// TIA Portal V21 export
FUNCTION "SUBOUT" : Void   // FC16, LAD
{ S7_Optimized_Access := 'TRUE' }
// stored: SetENOAutomatically false
   VAR_TEMP   // added for the SCL form of the ladder/FBD networks
      _w1 : Bool;
      _w2 : Bool;
   END_VAR
BEGIN

REGION Network 1
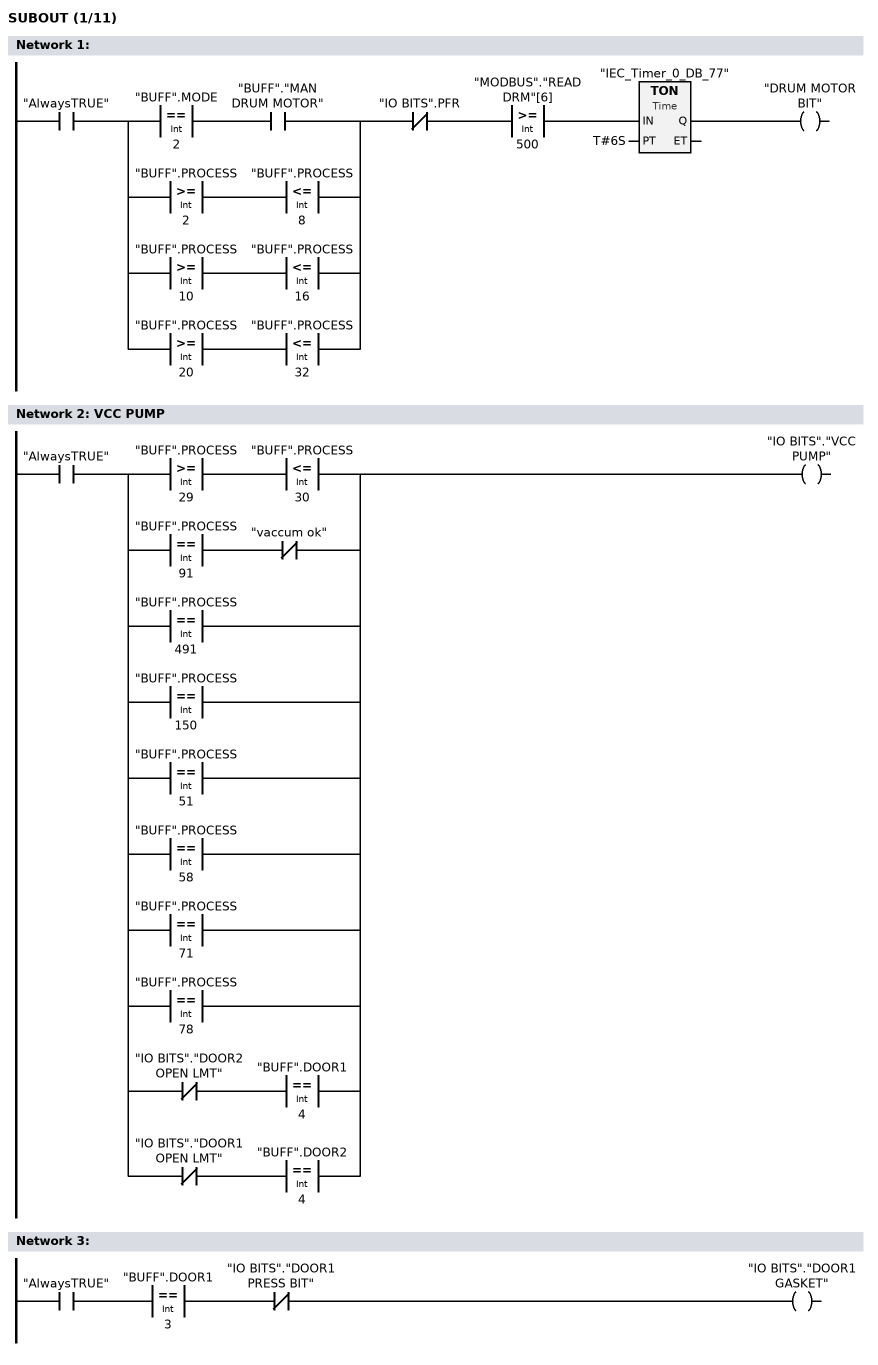
   RUNG wire#powerrail
      Contact( "AlwaysTRUE" )
      wire#w1
      { S7_Templates := "SrcType := Int" } EQ_Contact(in1 := "BUFF".MODE, in2 := 2)
      Contact( "BUFF"."MAN DRUM MOTOR" )
      wire#w2
      I_Contact( "IO BITS".PFR )
      { S7_Templates := "SrcType := Int" } GE_Contact(in1 := "MODBUS"."READ DRM"[6], in2 := 500)
      { S7_Templates := "time_type := Time" } "IEC_Timer_0_DB_77".TON(pt := T#6S, et =>)
      Coil( "DRUM MOTOR BIT" )
   END_RUNG
   RUNG wire#w1
      { S7_Templates := "SrcType := Int" } GE_Contact(in1 := "BUFF".PROCESS, in2 := 2)
      { S7_Templates := "SrcType := Int" } LE_Contact(in1 := "BUFF".PROCESS, in2 := 8)
   END_RUNG wire#w2
   RUNG wire#w1
      { S7_Templates := "SrcType := Int" } GE_Contact(in1 := "BUFF".PROCESS, in2 := 10)
      { S7_Templates := "SrcType := Int" } LE_Contact(in1 := "BUFF".PROCESS, in2 := 16)
   END_RUNG wire#w2
   RUNG wire#w1
      { S7_Templates := "SrcType := Int" } GE_Contact(in1 := "BUFF".PROCESS, in2 := 20)
      { S7_Templates := "SrcType := Int" } LE_Contact(in1 := "BUFF".PROCESS, in2 := 32)
   END_RUNG wire#w2
   // the same network as SCL:
   "IEC_Timer_0_DB_77".TON(IN := "AlwaysTRUE" AND ((("BUFF".MODE = 2) AND "BUFF"."MAN DRUM MOTOR") OR (("BUFF".PROCESS >= 2) AND ("BUFF".PROCESS <= 8)) OR (("BUFF".PROCESS >= 10) AND ("BUFF".PROCESS <= 16)) OR (("BUFF".PROCESS >= 20) AND ("BUFF".PROCESS <= 32))) AND NOT "IO BITS".PFR AND ("MODBUS"."READ DRM"[6] >= 500),
                           PT := T#6S);
   "DRUM MOTOR BIT" := "IEC_Timer_0_DB_77".Q;
END_REGION

REGION Network 2: VCC PUMP
   RUNG wire#powerrail
      Contact( "AlwaysTRUE" )
      wire#w1
      { S7_Templates := "SrcType := Int" } GE_Contact(in1 := "BUFF".PROCESS, in2 := 29)
      { S7_Templates := "SrcType := Int" } LE_Contact(in1 := "BUFF".PROCESS, in2 := 30)
      wire#w2
      Coil( "IO BITS"."VCC PUMP" )
   END_RUNG
   RUNG wire#w1
      { S7_Templates := "SrcType := Int" } EQ_Contact(in1 := "BUFF".PROCESS, in2 := 91)
      I_Contact( "vaccum ok" )
   END_RUNG wire#w2
   RUNG wire#w1
      { S7_Templates := "SrcType := Int" } EQ_Contact(in1 := "BUFF".PROCESS, in2 := 491)
   END_RUNG wire#w2
   RUNG wire#w1
      { S7_Templates := "SrcType := Int" } EQ_Contact(in1 := "BUFF".PROCESS, in2 := 150)
   END_RUNG wire#w2
   RUNG wire#w1
      { S7_Templates := "SrcType := Int" } EQ_Contact(in1 := "BUFF".PROCESS, in2 := 51)
   END_RUNG wire#w2
   RUNG wire#w1
      { S7_Templates := "SrcType := Int" } EQ_Contact(in1 := "BUFF".PROCESS, in2 := 58)
   END_RUNG wire#w2
   RUNG wire#w1
      { S7_Templates := "SrcType := Int" } EQ_Contact(in1 := "BUFF".PROCESS, in2 := 71)
   END_RUNG wire#w2
   RUNG wire#w1
      { S7_Templates := "SrcType := Int" } EQ_Contact(in1 := "BUFF".PROCESS, in2 := 78)
   END_RUNG wire#w2
   RUNG wire#w1
      I_Contact( "IO BITS"."DOOR2 OPEN LMT" )
      { S7_Templates := "SrcType := Int" } EQ_Contact(in1 := "BUFF".DOOR1, in2 := 4)
   END_RUNG wire#w2
   RUNG wire#w1
      I_Contact( "IO BITS"."DOOR1 OPEN LMT" )
      { S7_Templates := "SrcType := Int" } EQ_Contact(in1 := "BUFF".DOOR2, in2 := 4)
   END_RUNG wire#w2
   // the same network as SCL:
   "IO BITS"."VCC PUMP" := "AlwaysTRUE" AND ((("BUFF".PROCESS >= 29) AND ("BUFF".PROCESS <= 30)) OR (("BUFF".PROCESS = 91) AND NOT "vaccum ok") OR ("BUFF".PROCESS = 491) OR ("BUFF".PROCESS = 150) OR ("BUFF".PROCESS = 51) OR ("BUFF".PROCESS = 58) OR ("BUFF".PROCESS = 71) OR ("BUFF".PROCESS = 78) OR (NOT "IO BITS"."DOOR2 OPEN LMT" AND ("BUFF".DOOR1 = 4)) OR (NOT "IO BITS"."DOOR1 OPEN LMT" AND ("BUFF".DOOR2 = 4)));
END_REGION

REGION Network 3
   RUNG wire#powerrail
      Contact( "AlwaysTRUE" )
      { S7_Templates := "SrcType := Int" } EQ_Contact(in1 := "BUFF".DOOR1, in2 := 3)
      I_Contact( "IO BITS"."DOOR1 PRESS BIT" )
      Coil( "IO BITS"."DOOR1 GASKET" )
   END_RUNG
   // the same network as SCL:
   "IO BITS"."DOOR1 GASKET" := "AlwaysTRUE" AND ("BUFF".DOOR1 = 3) AND NOT "IO BITS"."DOOR1 PRESS BIT";
END_REGION

REGION Network 4
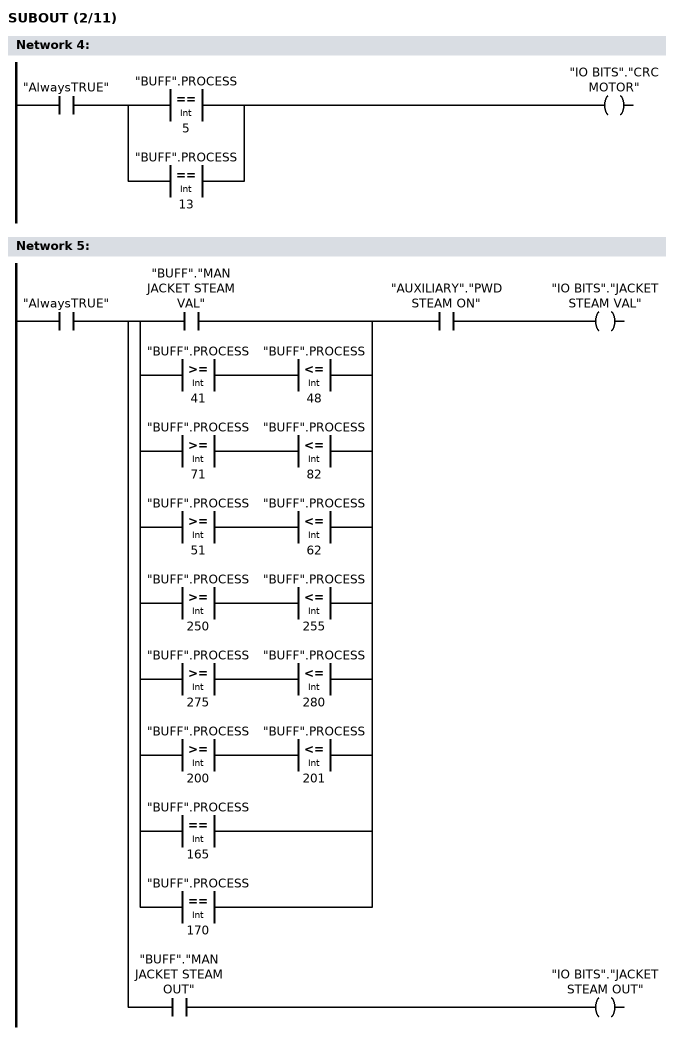
   RUNG wire#powerrail
      Contact( "AlwaysTRUE" )
      wire#w1
      { S7_Templates := "SrcType := Int" } EQ_Contact(in1 := "BUFF".PROCESS, in2 := 5)
      wire#w2
      Coil( "IO BITS"."CRC MOTOR" )
   END_RUNG
   RUNG wire#w1
      { S7_Templates := "SrcType := Int" } EQ_Contact(in1 := "BUFF".PROCESS, in2 := 13)
   END_RUNG wire#w2
   // the same network as SCL:
   "IO BITS"."CRC MOTOR" := "AlwaysTRUE" AND (("BUFF".PROCESS = 5) OR ("BUFF".PROCESS = 13));
END_REGION

REGION Network 5
   RUNG wire#powerrail
      Contact( "AlwaysTRUE" )
      wire#w1
      Contact( "BUFF"."MAN JACKET STEAM VAL" )
      wire#w2
      Contact( "AUXILIARY"."PWD STEAM ON" )
      Coil( "IO BITS"."JACKET STEAM VAL" )
   END_RUNG
   RUNG wire#w1
      { S7_Templates := "SrcType := Int" } GE_Contact(in1 := "BUFF".PROCESS, in2 := 41)
      { S7_Templates := "SrcType := Int" } LE_Contact(in1 := "BUFF".PROCESS, in2 := 48)
   END_RUNG wire#w2
   RUNG wire#w1
      { S7_Templates := "SrcType := Int" } GE_Contact(in1 := "BUFF".PROCESS, in2 := 71)
      { S7_Templates := "SrcType := Int" } LE_Contact(in1 := "BUFF".PROCESS, in2 := 82)
   END_RUNG wire#w2
   RUNG wire#w1
      { S7_Templates := "SrcType := Int" } GE_Contact(in1 := "BUFF".PROCESS, in2 := 51)
      { S7_Templates := "SrcType := Int" } LE_Contact(in1 := "BUFF".PROCESS, in2 := 62)
   END_RUNG wire#w2
   RUNG wire#w1
      { S7_Templates := "SrcType := Int" } GE_Contact(in1 := "BUFF".PROCESS, in2 := 250)
      { S7_Templates := "SrcType := Int" } LE_Contact(in1 := "BUFF".PROCESS, in2 := 255)
   END_RUNG wire#w2
   RUNG wire#w1
      { S7_Templates := "SrcType := Int" } GE_Contact(in1 := "BUFF".PROCESS, in2 := 275)
      { S7_Templates := "SrcType := Int" } LE_Contact(in1 := "BUFF".PROCESS, in2 := 280)
   END_RUNG wire#w2
   RUNG wire#w1
      { S7_Templates := "SrcType := Int" } GE_Contact(in1 := "BUFF".PROCESS, in2 := 200)
      { S7_Templates := "SrcType := Int" } LE_Contact(in1 := "BUFF".PROCESS, in2 := 201)
   END_RUNG wire#w2
   RUNG wire#w1
      { S7_Templates := "SrcType := Int" } EQ_Contact(in1 := "BUFF".PROCESS, in2 := 165)
   END_RUNG wire#w2
   RUNG wire#w1
      { S7_Templates := "SrcType := Int" } EQ_Contact(in1 := "BUFF".PROCESS, in2 := 170)
   END_RUNG wire#w2
   RUNG wire#w1
      Contact( "BUFF"."MAN JACKET STEAM OUT" )
      Coil( "IO BITS"."JACKET STEAM OUT" )
   END_RUNG
   // the same network as SCL:
   "IO BITS"."JACKET STEAM VAL" := "AlwaysTRUE" AND ("BUFF"."MAN JACKET STEAM VAL" OR (("BUFF".PROCESS >= 41) AND ("BUFF".PROCESS <= 48)) OR (("BUFF".PROCESS >= 71) AND ("BUFF".PROCESS <= 82)) OR (("BUFF".PROCESS >= 51) AND ("BUFF".PROCESS <= 62)) OR (("BUFF".PROCESS >= 250) AND ("BUFF".PROCESS <= 255)) OR (("BUFF".PROCESS >= 275) AND ("BUFF".PROCESS <= 280)) OR (("BUFF".PROCESS >= 200) AND ("BUFF".PROCESS <= 201)) OR ("BUFF".PROCESS = 165) OR ("BUFF".PROCESS = 170)) AND "AUXILIARY"."PWD STEAM ON";
   "IO BITS"."JACKET STEAM OUT" := "AlwaysTRUE" AND "BUFF"."MAN JACKET STEAM OUT";
END_REGION

REGION Network 6
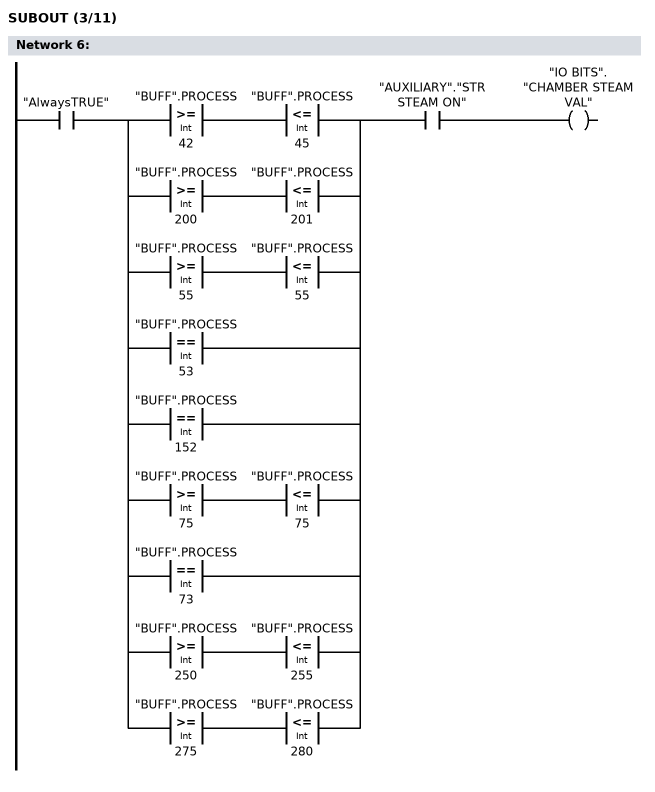
   RUNG wire#powerrail
      Contact( "AlwaysTRUE" )
      wire#w1
      { S7_Templates := "SrcType := Int" } GE_Contact(in1 := "BUFF".PROCESS, in2 := 42)
      { S7_Templates := "SrcType := Int" } LE_Contact(in1 := "BUFF".PROCESS, in2 := 45)
      wire#w2
      Contact( "AUXILIARY"."STR STEAM ON" )
      Coil( "IO BITS"."CHAMBER STEAM VAL" )
   END_RUNG
   RUNG wire#w1
      { S7_Templates := "SrcType := Int" } GE_Contact(in1 := "BUFF".PROCESS, in2 := 200)
      { S7_Templates := "SrcType := Int" } LE_Contact(in1 := "BUFF".PROCESS, in2 := 201)
   END_RUNG wire#w2
   RUNG wire#w1
      { S7_Templates := "SrcType := Int" } GE_Contact(in1 := "BUFF".PROCESS, in2 := 55)
      { S7_Templates := "SrcType := Int" } LE_Contact(in1 := "BUFF".PROCESS, in2 := 55)
   END_RUNG wire#w2
   RUNG wire#w1
      { S7_Templates := "SrcType := Int" } EQ_Contact(in1 := "BUFF".PROCESS, in2 := 53)
   END_RUNG wire#w2
   RUNG wire#w1
      { S7_Templates := "SrcType := Int" } EQ_Contact(in1 := "BUFF".PROCESS, in2 := 152)
   END_RUNG wire#w2
   RUNG wire#w1
      { S7_Templates := "SrcType := Int" } GE_Contact(in1 := "BUFF".PROCESS, in2 := 75)
      { S7_Templates := "SrcType := Int" } LE_Contact(in1 := "BUFF".PROCESS, in2 := 75)
   END_RUNG wire#w2
   RUNG wire#w1
      { S7_Templates := "SrcType := Int" } EQ_Contact(in1 := "BUFF".PROCESS, in2 := 73)
   END_RUNG wire#w2
   RUNG wire#w1
      { S7_Templates := "SrcType := Int" } GE_Contact(in1 := "BUFF".PROCESS, in2 := 250)
      { S7_Templates := "SrcType := Int" } LE_Contact(in1 := "BUFF".PROCESS, in2 := 255)
   END_RUNG wire#w2
   RUNG wire#w1
      { S7_Templates := "SrcType := Int" } GE_Contact(in1 := "BUFF".PROCESS, in2 := 275)
      { S7_Templates := "SrcType := Int" } LE_Contact(in1 := "BUFF".PROCESS, in2 := 280)
   END_RUNG wire#w2
   // the same network as SCL:
   "IO BITS"."CHAMBER STEAM VAL" := "AlwaysTRUE" AND ((("BUFF".PROCESS >= 42) AND ("BUFF".PROCESS <= 45)) OR (("BUFF".PROCESS >= 200) AND ("BUFF".PROCESS <= 201)) OR (("BUFF".PROCESS >= 55) AND ("BUFF".PROCESS <= 55)) OR ("BUFF".PROCESS = 53) OR ("BUFF".PROCESS = 152) OR (("BUFF".PROCESS >= 75) AND ("BUFF".PROCESS <= 75)) OR ("BUFF".PROCESS = 73) OR (("BUFF".PROCESS >= 250) AND ("BUFF".PROCESS <= 255)) OR (("BUFF".PROCESS >= 275) AND ("BUFF".PROCESS <= 280))) AND "AUXILIARY"."STR STEAM ON";
END_REGION

REGION Network 7: CHAMBER EXHAUST VAL
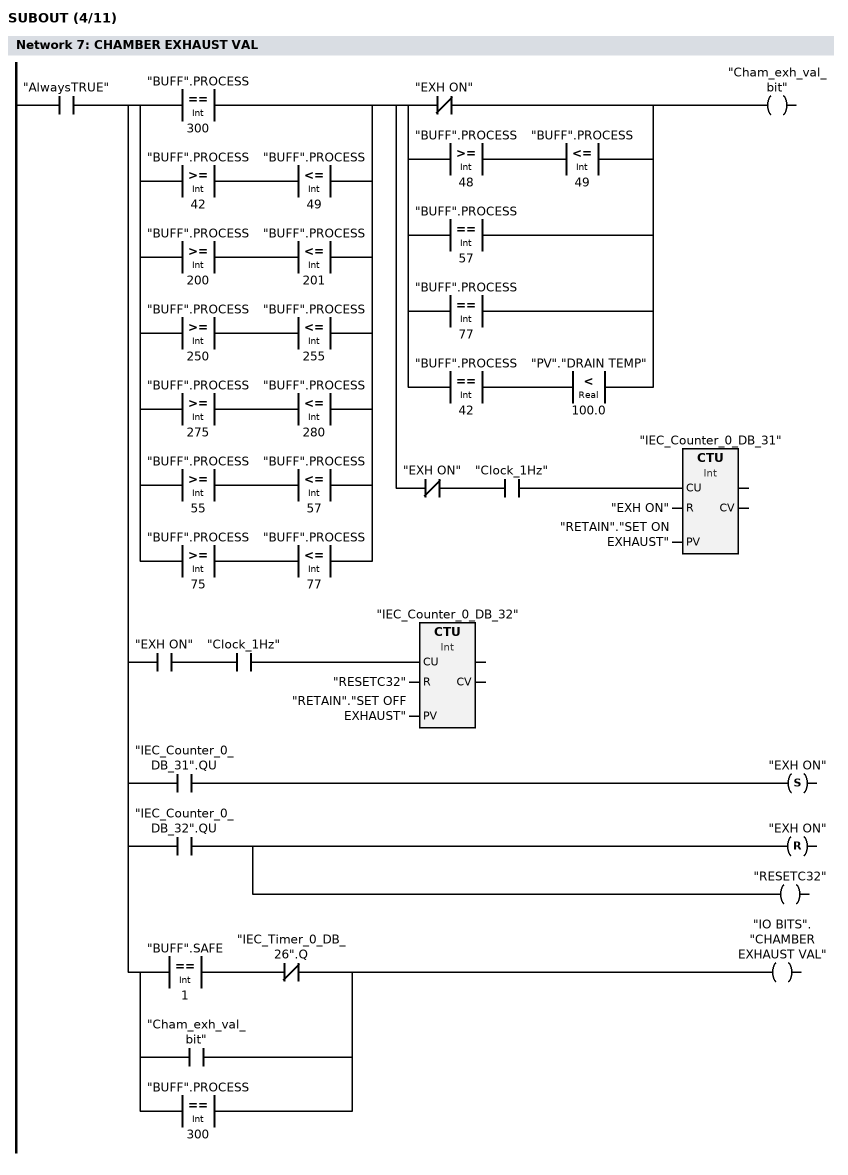
   RUNG wire#powerrail
      Contact( "AlwaysTRUE" )
      wire#w1
      { S7_Templates := "SrcType := Int" } EQ_Contact(in1 := "BUFF".PROCESS, in2 := 300)
      wire#w2
      I_Contact( "EXH ON" )
      wire#w3
      Coil( "Cham_exh_val_bit" )
   END_RUNG
   RUNG wire#w1
      { S7_Templates := "SrcType := Int" } GE_Contact(in1 := "BUFF".PROCESS, in2 := 42)
      { S7_Templates := "SrcType := Int" } LE_Contact(in1 := "BUFF".PROCESS, in2 := 49)
   END_RUNG wire#w2
   RUNG wire#w1
      { S7_Templates := "SrcType := Int" } GE_Contact(in1 := "BUFF".PROCESS, in2 := 200)
      { S7_Templates := "SrcType := Int" } LE_Contact(in1 := "BUFF".PROCESS, in2 := 201)
   END_RUNG wire#w2
   RUNG wire#w1
      { S7_Templates := "SrcType := Int" } GE_Contact(in1 := "BUFF".PROCESS, in2 := 250)
      { S7_Templates := "SrcType := Int" } LE_Contact(in1 := "BUFF".PROCESS, in2 := 255)
   END_RUNG wire#w2
   RUNG wire#w1
      { S7_Templates := "SrcType := Int" } GE_Contact(in1 := "BUFF".PROCESS, in2 := 275)
      { S7_Templates := "SrcType := Int" } LE_Contact(in1 := "BUFF".PROCESS, in2 := 280)
   END_RUNG wire#w2
   RUNG wire#w1
      { S7_Templates := "SrcType := Int" } GE_Contact(in1 := "BUFF".PROCESS, in2 := 55)
      { S7_Templates := "SrcType := Int" } LE_Contact(in1 := "BUFF".PROCESS, in2 := 57)
   END_RUNG wire#w2
   RUNG wire#w1
      { S7_Templates := "SrcType := Int" } GE_Contact(in1 := "BUFF".PROCESS, in2 := 75)
      { S7_Templates := "SrcType := Int" } LE_Contact(in1 := "BUFF".PROCESS, in2 := 77)
   END_RUNG wire#w2
   RUNG wire#w2
      { S7_Templates := "SrcType := Int" } GE_Contact(in1 := "BUFF".PROCESS, in2 := 48)
      { S7_Templates := "SrcType := Int" } LE_Contact(in1 := "BUFF".PROCESS, in2 := 49)
   END_RUNG wire#w3
   RUNG wire#w2
      { S7_Templates := "SrcType := Int" } EQ_Contact(in1 := "BUFF".PROCESS, in2 := 57)
   END_RUNG wire#w3
   RUNG wire#w2
      { S7_Templates := "SrcType := Int" } EQ_Contact(in1 := "BUFF".PROCESS, in2 := 77)
   END_RUNG wire#w3
   RUNG wire#w2
      { S7_Templates := "SrcType := Int" } EQ_Contact(in1 := "BUFF".PROCESS, in2 := 42)
      { S7_Templates := "SrcType := Real" } LT_Contact(in1 := "PV"."DRAIN TEMP", in2 := 100.0)
   END_RUNG wire#w3
   RUNG wire#w2
      I_Contact( "EXH ON" )
      Contact( "Clock_1Hz" )
      { S7_Templates := "value_type := Int" } "IEC_Counter_0_DB_31".CTU(r := "EXH ON", pv := "RETAIN"."SET ON EXHAUST", cv =>)
   END_RUNG
   RUNG wire#w1
      Contact( "EXH ON" )
      Contact( "Clock_1Hz" )
      { S7_Templates := "value_type := Int" } "IEC_Counter_0_DB_32".CTU(r := "RESETC32", pv := "RETAIN"."SET OFF EXHAUST", cv =>)
   END_RUNG
   RUNG wire#w1
      Contact( "IEC_Counter_0_DB_31".QU )
      S_Coil( "EXH ON" )
   END_RUNG
   RUNG wire#w1
      Contact( "IEC_Counter_0_DB_32".QU )
      wire#w4
      R_Coil( "EXH ON" )
   END_RUNG
   RUNG wire#w4
      Coil( "RESETC32" )
   END_RUNG
   RUNG wire#w1
      { S7_Templates := "SrcType := Int" } EQ_Contact(in1 := "BUFF".SAFE, in2 := 1)
      I_Contact( "IEC_Timer_0_DB_26".Q )
      wire#w5
      Coil( "IO BITS"."CHAMBER EXHAUST VAL" )
   END_RUNG
   RUNG wire#w1
      Contact( "Cham_exh_val_bit" )
   END_RUNG wire#w5
   RUNG wire#w1
      { S7_Templates := "SrcType := Int" } EQ_Contact(in1 := "BUFF".PROCESS, in2 := 300)
   END_RUNG wire#w5
   // the same network as SCL:
   #_w1 := "AlwaysTRUE" AND (("BUFF".PROCESS = 300) OR (("BUFF".PROCESS >= 42) AND ("BUFF".PROCESS <= 49)) OR (("BUFF".PROCESS >= 200) AND ("BUFF".PROCESS <= 201)) OR (("BUFF".PROCESS >= 250) AND ("BUFF".PROCESS <= 255)) OR (("BUFF".PROCESS >= 275) AND ("BUFF".PROCESS <= 280)) OR (("BUFF".PROCESS >= 55) AND ("BUFF".PROCESS <= 57)) OR (("BUFF".PROCESS >= 75) AND ("BUFF".PROCESS <= 77)));
   "Cham_exh_val_bit" := #_w1 AND (NOT "EXH ON" OR (("BUFF".PROCESS >= 48) AND ("BUFF".PROCESS <= 49)) OR ("BUFF".PROCESS = 57) OR ("BUFF".PROCESS = 77) OR (("BUFF".PROCESS = 42) AND ("PV"."DRAIN TEMP" < 100.0)));
   "IEC_Counter_0_DB_31".CTU(CU := #_w1 AND NOT "EXH ON" AND "Clock_1Hz",
                           R := "EXH ON",
                           PV := "RETAIN"."SET ON EXHAUST");
   "IEC_Counter_0_DB_32".CTU(CU := "AlwaysTRUE" AND "EXH ON" AND "Clock_1Hz",
                           R := "RESETC32",
                           PV := "RETAIN"."SET OFF EXHAUST");
   IF "AlwaysTRUE" AND "IEC_Counter_0_DB_31".QU THEN "EXH ON" := TRUE; END_IF;
   #_w2 := "AlwaysTRUE" AND "IEC_Counter_0_DB_32".QU;
   IF #_w2 THEN "EXH ON" := FALSE; END_IF;
   "RESETC32" := #_w2;
   "IO BITS"."CHAMBER EXHAUST VAL" := "AlwaysTRUE" AND ((("BUFF".SAFE = 1) AND NOT "IEC_Timer_0_DB_26".Q) OR "Cham_exh_val_bit" OR ("BUFF".PROCESS = 300));
END_REGION

REGION Network 8
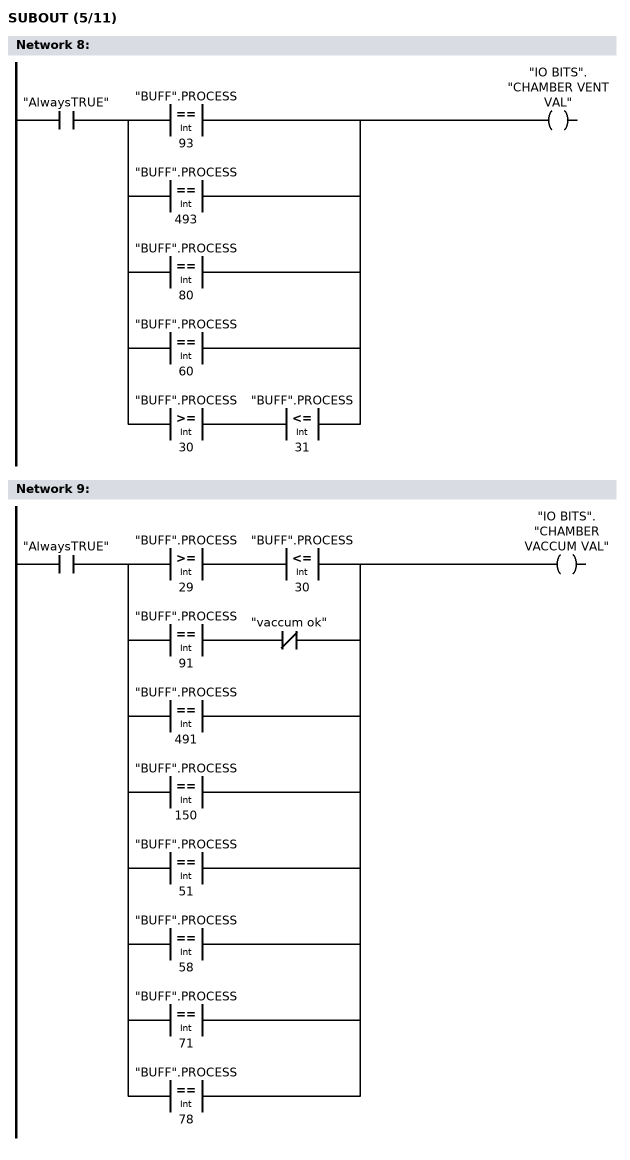
   RUNG wire#powerrail
      Contact( "AlwaysTRUE" )
      wire#w1
      { S7_Templates := "SrcType := Int" } EQ_Contact(in1 := "BUFF".PROCESS, in2 := 93)
      wire#w2
      Coil( "IO BITS"."CHAMBER VENT VAL" )
   END_RUNG
   RUNG wire#w1
      { S7_Templates := "SrcType := Int" } EQ_Contact(in1 := "BUFF".PROCESS, in2 := 493)
   END_RUNG wire#w2
   RUNG wire#w1
      { S7_Templates := "SrcType := Int" } EQ_Contact(in1 := "BUFF".PROCESS, in2 := 80)
   END_RUNG wire#w2
   RUNG wire#w1
      { S7_Templates := "SrcType := Int" } EQ_Contact(in1 := "BUFF".PROCESS, in2 := 60)
   END_RUNG wire#w2
   RUNG wire#w1
      { S7_Templates := "SrcType := Int" } GE_Contact(in1 := "BUFF".PROCESS, in2 := 30)
      { S7_Templates := "SrcType := Int" } LE_Contact(in1 := "BUFF".PROCESS, in2 := 31)
   END_RUNG wire#w2
   // the same network as SCL:
   "IO BITS"."CHAMBER VENT VAL" := "AlwaysTRUE" AND (("BUFF".PROCESS = 93) OR ("BUFF".PROCESS = 493) OR ("BUFF".PROCESS = 80) OR ("BUFF".PROCESS = 60) OR (("BUFF".PROCESS >= 30) AND ("BUFF".PROCESS <= 31)));
END_REGION

REGION Network 9
   RUNG wire#powerrail
      Contact( "AlwaysTRUE" )
      wire#w1
      { S7_Templates := "SrcType := Int" } GE_Contact(in1 := "BUFF".PROCESS, in2 := 29)
      { S7_Templates := "SrcType := Int" } LE_Contact(in1 := "BUFF".PROCESS, in2 := 30)
      wire#w2
      Coil( "IO BITS"."CHAMBER VACCUM VAL" )
   END_RUNG
   RUNG wire#w1
      { S7_Templates := "SrcType := Int" } EQ_Contact(in1 := "BUFF".PROCESS, in2 := 91)
      I_Contact( "vaccum ok" )
   END_RUNG wire#w2
   RUNG wire#w1
      { S7_Templates := "SrcType := Int" } EQ_Contact(in1 := "BUFF".PROCESS, in2 := 491)
   END_RUNG wire#w2
   RUNG wire#w1
      { S7_Templates := "SrcType := Int" } EQ_Contact(in1 := "BUFF".PROCESS, in2 := 150)
   END_RUNG wire#w2
   RUNG wire#w1
      { S7_Templates := "SrcType := Int" } EQ_Contact(in1 := "BUFF".PROCESS, in2 := 51)
   END_RUNG wire#w2
   RUNG wire#w1
      { S7_Templates := "SrcType := Int" } EQ_Contact(in1 := "BUFF".PROCESS, in2 := 58)
   END_RUNG wire#w2
   RUNG wire#w1
      { S7_Templates := "SrcType := Int" } EQ_Contact(in1 := "BUFF".PROCESS, in2 := 71)
   END_RUNG wire#w2
   RUNG wire#w1
      { S7_Templates := "SrcType := Int" } EQ_Contact(in1 := "BUFF".PROCESS, in2 := 78)
   END_RUNG wire#w2
   // the same network as SCL:
   "IO BITS"."CHAMBER VACCUM VAL" := "AlwaysTRUE" AND ((("BUFF".PROCESS >= 29) AND ("BUFF".PROCESS <= 30)) OR (("BUFF".PROCESS = 91) AND NOT "vaccum ok") OR ("BUFF".PROCESS = 491) OR ("BUFF".PROCESS = 150) OR ("BUFF".PROCESS = 51) OR ("BUFF".PROCESS = 58) OR ("BUFF".PROCESS = 71) OR ("BUFF".PROCESS = 78));
END_REGION

REGION Network 10
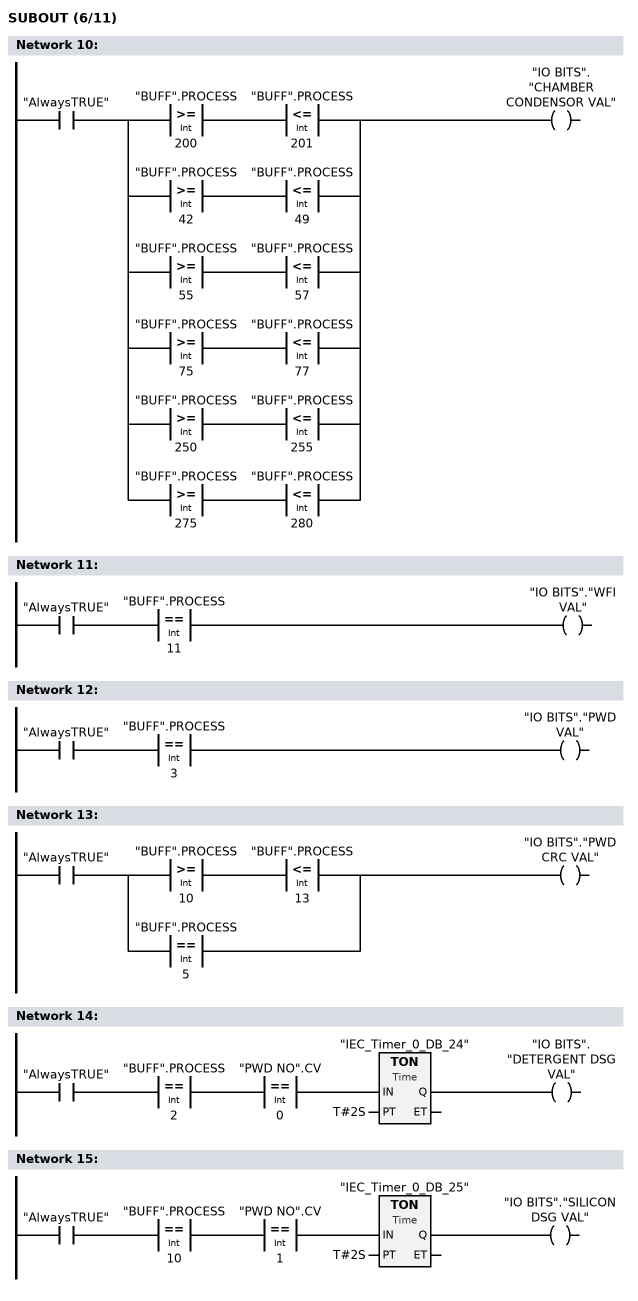
   RUNG wire#powerrail
      Contact( "AlwaysTRUE" )
      wire#w1
      { S7_Templates := "SrcType := Int" } GE_Contact(in1 := "BUFF".PROCESS, in2 := 200)
      { S7_Templates := "SrcType := Int" } LE_Contact(in1 := "BUFF".PROCESS, in2 := 201)
      wire#w2
      Coil( "IO BITS"."CHAMBER CONDENSOR VAL" )
   END_RUNG
   RUNG wire#w1
      { S7_Templates := "SrcType := Int" } GE_Contact(in1 := "BUFF".PROCESS, in2 := 42)
      { S7_Templates := "SrcType := Int" } LE_Contact(in1 := "BUFF".PROCESS, in2 := 49)
   END_RUNG wire#w2
   RUNG wire#w1
      { S7_Templates := "SrcType := Int" } GE_Contact(in1 := "BUFF".PROCESS, in2 := 55)
      { S7_Templates := "SrcType := Int" } LE_Contact(in1 := "BUFF".PROCESS, in2 := 57)
   END_RUNG wire#w2
   RUNG wire#w1
      { S7_Templates := "SrcType := Int" } GE_Contact(in1 := "BUFF".PROCESS, in2 := 75)
      { S7_Templates := "SrcType := Int" } LE_Contact(in1 := "BUFF".PROCESS, in2 := 77)
   END_RUNG wire#w2
   RUNG wire#w1
      { S7_Templates := "SrcType := Int" } GE_Contact(in1 := "BUFF".PROCESS, in2 := 250)
      { S7_Templates := "SrcType := Int" } LE_Contact(in1 := "BUFF".PROCESS, in2 := 255)
   END_RUNG wire#w2
   RUNG wire#w1
      { S7_Templates := "SrcType := Int" } GE_Contact(in1 := "BUFF".PROCESS, in2 := 275)
      { S7_Templates := "SrcType := Int" } LE_Contact(in1 := "BUFF".PROCESS, in2 := 280)
   END_RUNG wire#w2
   // the same network as SCL:
   "IO BITS"."CHAMBER CONDENSOR VAL" := "AlwaysTRUE" AND ((("BUFF".PROCESS >= 200) AND ("BUFF".PROCESS <= 201)) OR (("BUFF".PROCESS >= 42) AND ("BUFF".PROCESS <= 49)) OR (("BUFF".PROCESS >= 55) AND ("BUFF".PROCESS <= 57)) OR (("BUFF".PROCESS >= 75) AND ("BUFF".PROCESS <= 77)) OR (("BUFF".PROCESS >= 250) AND ("BUFF".PROCESS <= 255)) OR (("BUFF".PROCESS >= 275) AND ("BUFF".PROCESS <= 280)));
END_REGION

REGION Network 11
   RUNG wire#powerrail
      Contact( "AlwaysTRUE" )
      { S7_Templates := "SrcType := Int" } EQ_Contact(in1 := "BUFF".PROCESS, in2 := 11)
      Coil( "IO BITS"."WFI VAL" )
   END_RUNG
   // the same network as SCL:
   "IO BITS"."WFI VAL" := "AlwaysTRUE" AND ("BUFF".PROCESS = 11);
END_REGION

REGION Network 12
   RUNG wire#powerrail
      Contact( "AlwaysTRUE" )
      { S7_Templates := "SrcType := Int" } EQ_Contact(in1 := "BUFF".PROCESS, in2 := 3)
      Coil( "IO BITS"."PWD VAL" )
   END_RUNG
   // the same network as SCL:
   "IO BITS"."PWD VAL" := "AlwaysTRUE" AND ("BUFF".PROCESS = 3);
END_REGION

REGION Network 13
   RUNG wire#powerrail
      Contact( "AlwaysTRUE" )
      wire#w1
      { S7_Templates := "SrcType := Int" } GE_Contact(in1 := "BUFF".PROCESS, in2 := 10)
      { S7_Templates := "SrcType := Int" } LE_Contact(in1 := "BUFF".PROCESS, in2 := 13)
      wire#w2
      Coil( "IO BITS"."PWD CRC VAL" )
   END_RUNG
   RUNG wire#w1
      { S7_Templates := "SrcType := Int" } EQ_Contact(in1 := "BUFF".PROCESS, in2 := 5)
   END_RUNG wire#w2
   // the same network as SCL:
   "IO BITS"."PWD CRC VAL" := "AlwaysTRUE" AND ((("BUFF".PROCESS >= 10) AND ("BUFF".PROCESS <= 13)) OR ("BUFF".PROCESS = 5));
END_REGION

REGION Network 14
   RUNG wire#powerrail
      Contact( "AlwaysTRUE" )
      { S7_Templates := "SrcType := Int" } EQ_Contact(in1 := "BUFF".PROCESS, in2 := 2)
      { S7_Templates := "SrcType := Int" } EQ_Contact(in1 := "PWD NO".CV, in2 := 0)
      { S7_Templates := "time_type := Time" } "IEC_Timer_0_DB_24".TON(pt := T#2S, et =>)
      Coil( "IO BITS"."DETERGENT DSG VAL" )
   END_RUNG
   // the same network as SCL:
   "IEC_Timer_0_DB_24".TON(IN := "AlwaysTRUE" AND ("BUFF".PROCESS = 2) AND ("PWD NO".CV = 0), PT := T#2S);
   "IO BITS"."DETERGENT DSG VAL" := "IEC_Timer_0_DB_24".Q;
END_REGION

REGION Network 15
   RUNG wire#powerrail
      Contact( "AlwaysTRUE" )
      { S7_Templates := "SrcType := Int" } EQ_Contact(in1 := "BUFF".PROCESS, in2 := 10)
      { S7_Templates := "SrcType := Int" } EQ_Contact(in1 := "PWD NO".CV, in2 := 1)
      { S7_Templates := "time_type := Time" } "IEC_Timer_0_DB_25".TON(pt := T#2S, et =>)
      Coil( "IO BITS"."SILICON DSG VAL" )
   END_RUNG
   // the same network as SCL:
   "IEC_Timer_0_DB_25".TON(IN := "AlwaysTRUE" AND ("BUFF".PROCESS = 10) AND ("PWD NO".CV = 1), PT := T#2S);
   "IO BITS"."SILICON DSG VAL" := "IEC_Timer_0_DB_25".Q;
END_REGION

REGION Network 16: DRAIN VAL
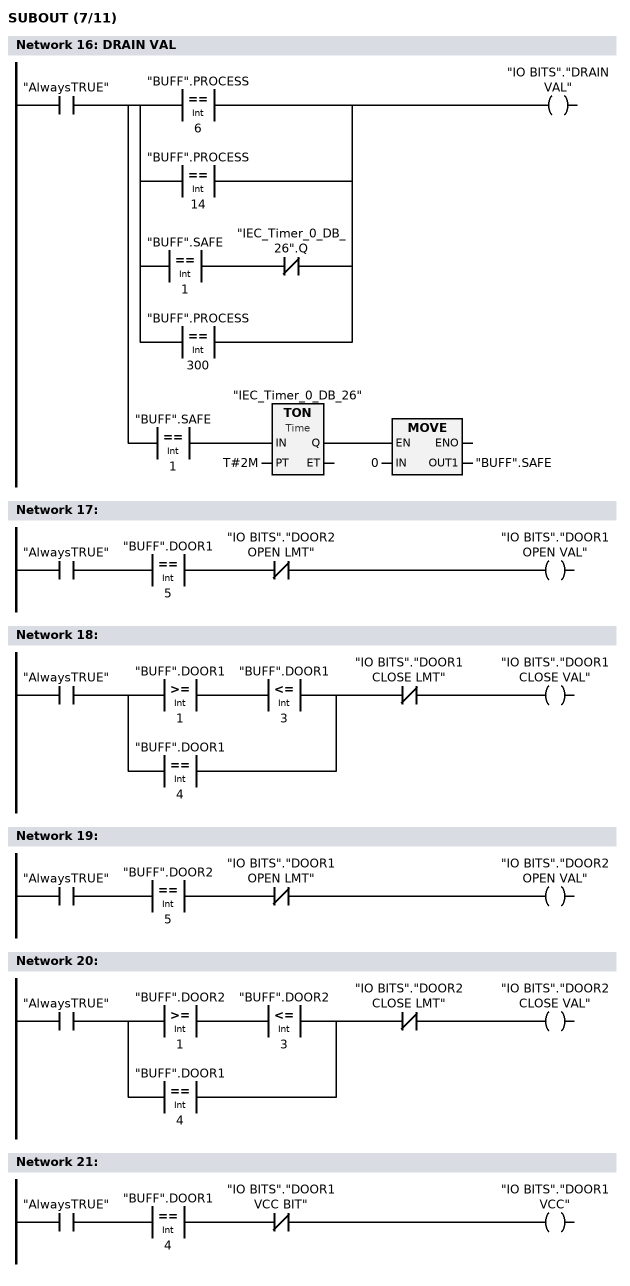
   RUNG wire#powerrail
      Contact( "AlwaysTRUE" )
      wire#w1
      { S7_Templates := "SrcType := Int" } EQ_Contact(in1 := "BUFF".PROCESS, in2 := 6)
      wire#w2
      Coil( "IO BITS"."DRAIN VAL" )
   END_RUNG
   RUNG wire#w1
      { S7_Templates := "SrcType := Int" } EQ_Contact(in1 := "BUFF".PROCESS, in2 := 14)
   END_RUNG wire#w2
   RUNG wire#w1
      { S7_Templates := "SrcType := Int" } EQ_Contact(in1 := "BUFF".SAFE, in2 := 1)
      I_Contact( "IEC_Timer_0_DB_26".Q )
   END_RUNG wire#w2
   RUNG wire#w1
      { S7_Templates := "SrcType := Int" } EQ_Contact(in1 := "BUFF".PROCESS, in2 := 300)
   END_RUNG wire#w2
   RUNG wire#w1
      { S7_Templates := "SrcType := Int" } EQ_Contact(in1 := "BUFF".SAFE, in2 := 1)
      { S7_Templates := "time_type := Time" } "IEC_Timer_0_DB_26".TON(pt := T#2M, et =>)
      Move(in := 0, out1 => "BUFF".SAFE)
   END_RUNG
   // the same network as SCL:
   "IO BITS"."DRAIN VAL" := "AlwaysTRUE" AND (("BUFF".PROCESS = 6) OR ("BUFF".PROCESS = 14) OR (("BUFF".SAFE = 1) AND NOT "IEC_Timer_0_DB_26".Q) OR ("BUFF".PROCESS = 300));
   "IEC_Timer_0_DB_26".TON(IN := "AlwaysTRUE" AND ("BUFF".SAFE = 1), PT := T#2M);
   IF "IEC_Timer_0_DB_26".Q THEN "BUFF".SAFE := 0; END_IF;
END_REGION

REGION Network 17
   RUNG wire#powerrail
      Contact( "AlwaysTRUE" )
      { S7_Templates := "SrcType := Int" } EQ_Contact(in1 := "BUFF".DOOR1, in2 := 5)
      I_Contact( "IO BITS"."DOOR2 OPEN LMT" )
      Coil( "IO BITS"."DOOR1 OPEN VAL" )
   END_RUNG
   // the same network as SCL:
   "IO BITS"."DOOR1 OPEN VAL" := "AlwaysTRUE" AND ("BUFF".DOOR1 = 5) AND NOT "IO BITS"."DOOR2 OPEN LMT";
END_REGION

REGION Network 18
   RUNG wire#powerrail
      Contact( "AlwaysTRUE" )
      wire#w1
      { S7_Templates := "SrcType := Int" } GE_Contact(in1 := "BUFF".DOOR1, in2 := 1)
      { S7_Templates := "SrcType := Int" } LE_Contact(in1 := "BUFF".DOOR1, in2 := 3)
      wire#w2
      I_Contact( "IO BITS"."DOOR1 CLOSE LMT" )
      Coil( "IO BITS"."DOOR1 CLOSE VAL" )
   END_RUNG
   RUNG wire#w1
      { S7_Templates := "SrcType := Int" } EQ_Contact(in1 := "BUFF".DOOR1, in2 := 4)
   END_RUNG wire#w2
   // the same network as SCL:
   "IO BITS"."DOOR1 CLOSE VAL" := "AlwaysTRUE" AND ((("BUFF".DOOR1 >= 1) AND ("BUFF".DOOR1 <= 3)) OR ("BUFF".DOOR1 = 4)) AND NOT "IO BITS"."DOOR1 CLOSE LMT";
END_REGION

REGION Network 19
   RUNG wire#powerrail
      Contact( "AlwaysTRUE" )
      { S7_Templates := "SrcType := Int" } EQ_Contact(in1 := "BUFF".DOOR2, in2 := 5)
      I_Contact( "IO BITS"."DOOR1 OPEN LMT" )
      Coil( "IO BITS"."DOOR2 OPEN VAL" )
   END_RUNG
   // the same network as SCL:
   "IO BITS"."DOOR2 OPEN VAL" := "AlwaysTRUE" AND ("BUFF".DOOR2 = 5) AND NOT "IO BITS"."DOOR1 OPEN LMT";
END_REGION

REGION Network 20
   RUNG wire#powerrail
      Contact( "AlwaysTRUE" )
      wire#w1
      { S7_Templates := "SrcType := Int" } GE_Contact(in1 := "BUFF".DOOR2, in2 := 1)
      { S7_Templates := "SrcType := Int" } LE_Contact(in1 := "BUFF".DOOR2, in2 := 3)
      wire#w2
      I_Contact( "IO BITS"."DOOR2 CLOSE LMT" )
      Coil( "IO BITS"."DOOR2 CLOSE VAL" )
   END_RUNG
   RUNG wire#w1
      { S7_Templates := "SrcType := Int" } EQ_Contact(in1 := "BUFF".DOOR1, in2 := 4)
   END_RUNG wire#w2
   // the same network as SCL:
   "IO BITS"."DOOR2 CLOSE VAL" := "AlwaysTRUE" AND ((("BUFF".DOOR2 >= 1) AND ("BUFF".DOOR2 <= 3)) OR ("BUFF".DOOR1 = 4)) AND NOT "IO BITS"."DOOR2 CLOSE LMT";
END_REGION

REGION Network 21
   RUNG wire#powerrail
      Contact( "AlwaysTRUE" )
      { S7_Templates := "SrcType := Int" } EQ_Contact(in1 := "BUFF".DOOR1, in2 := 4)
      I_Contact( "IO BITS"."DOOR1 VCC BIT" )
      Coil( "IO BITS"."DOOR1 VCC" )
   END_RUNG
   // the same network as SCL:
   "IO BITS"."DOOR1 VCC" := "AlwaysTRUE" AND ("BUFF".DOOR1 = 4) AND NOT "IO BITS"."DOOR1 VCC BIT";
END_REGION

REGION Network 22
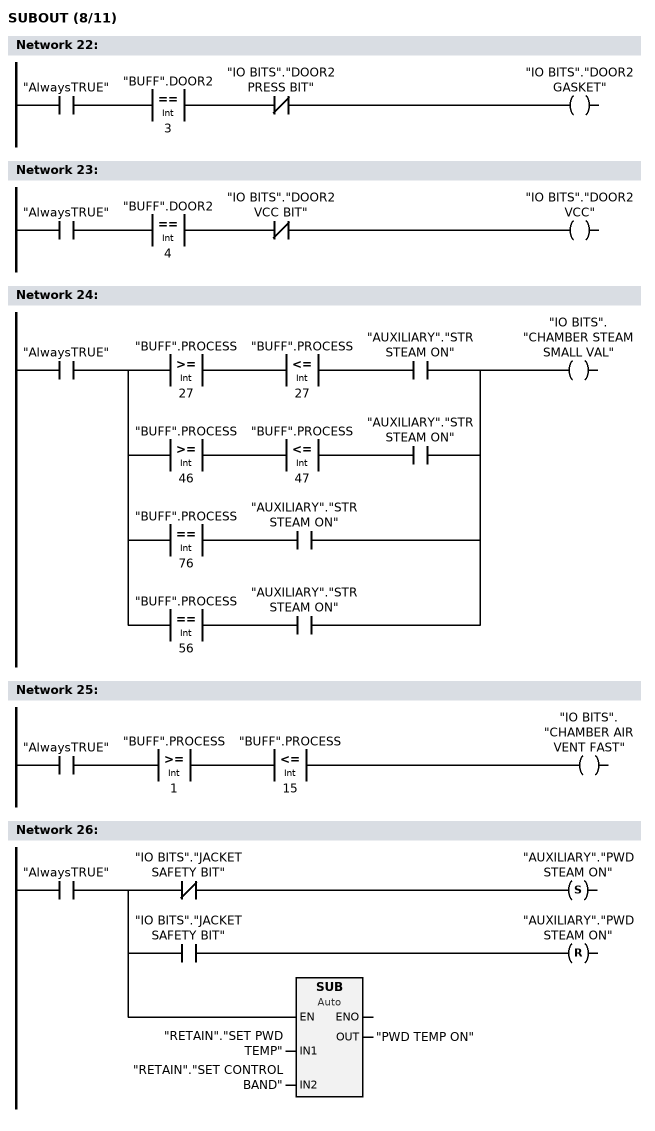
   RUNG wire#powerrail
      Contact( "AlwaysTRUE" )
      { S7_Templates := "SrcType := Int" } EQ_Contact(in1 := "BUFF".DOOR2, in2 := 3)
      I_Contact( "IO BITS"."DOOR2 PRESS BIT" )
      Coil( "IO BITS"."DOOR2 GASKET" )
   END_RUNG
   // the same network as SCL:
   "IO BITS"."DOOR2 GASKET" := "AlwaysTRUE" AND ("BUFF".DOOR2 = 3) AND NOT "IO BITS"."DOOR2 PRESS BIT";
END_REGION

REGION Network 23
   RUNG wire#powerrail
      Contact( "AlwaysTRUE" )
      { S7_Templates := "SrcType := Int" } EQ_Contact(in1 := "BUFF".DOOR2, in2 := 4)
      I_Contact( "IO BITS"."DOOR2 VCC BIT" )
      Coil( "IO BITS"."DOOR2 VCC" )
   END_RUNG
   // the same network as SCL:
   "IO BITS"."DOOR2 VCC" := "AlwaysTRUE" AND ("BUFF".DOOR2 = 4) AND NOT "IO BITS"."DOOR2 VCC BIT";
END_REGION

REGION Network 24
   RUNG wire#powerrail
      Contact( "AlwaysTRUE" )
      wire#w1
      { S7_Templates := "SrcType := Int" } GE_Contact(in1 := "BUFF".PROCESS, in2 := 27)
      { S7_Templates := "SrcType := Int" } LE_Contact(in1 := "BUFF".PROCESS, in2 := 27)
      Contact( "AUXILIARY"."STR STEAM ON" )
      wire#w2
      Coil( "IO BITS"."CHAMBER STEAM SMALL VAL" )
   END_RUNG
   RUNG wire#w1
      { S7_Templates := "SrcType := Int" } GE_Contact(in1 := "BUFF".PROCESS, in2 := 46)
      { S7_Templates := "SrcType := Int" } LE_Contact(in1 := "BUFF".PROCESS, in2 := 47)
      Contact( "AUXILIARY"."STR STEAM ON" )
   END_RUNG wire#w2
   RUNG wire#w1
      { S7_Templates := "SrcType := Int" } EQ_Contact(in1 := "BUFF".PROCESS, in2 := 76)
      Contact( "AUXILIARY"."STR STEAM ON" )
   END_RUNG wire#w2
   RUNG wire#w1
      { S7_Templates := "SrcType := Int" } EQ_Contact(in1 := "BUFF".PROCESS, in2 := 56)
      Contact( "AUXILIARY"."STR STEAM ON" )
   END_RUNG wire#w2
   // the same network as SCL:
   "IO BITS"."CHAMBER STEAM SMALL VAL" := "AlwaysTRUE" AND ((("BUFF".PROCESS >= 27) AND ("BUFF".PROCESS <= 27) AND "AUXILIARY"."STR STEAM ON") OR (("BUFF".PROCESS >= 46) AND ("BUFF".PROCESS <= 47) AND "AUXILIARY"."STR STEAM ON") OR (("BUFF".PROCESS = 76) AND "AUXILIARY"."STR STEAM ON") OR (("BUFF".PROCESS = 56) AND "AUXILIARY"."STR STEAM ON"));
END_REGION

REGION Network 25
   RUNG wire#powerrail
      Contact( "AlwaysTRUE" )
      { S7_Templates := "SrcType := Int" } GE_Contact(in1 := "BUFF".PROCESS, in2 := 1)
      { S7_Templates := "SrcType := Int" } LE_Contact(in1 := "BUFF".PROCESS, in2 := 15)
      Coil( "IO BITS"."CHAMBER AIR VENT FAST" )
   END_RUNG
   // the same network as SCL:
   "IO BITS"."CHAMBER AIR VENT FAST" := "AlwaysTRUE" AND ("BUFF".PROCESS >= 1) AND ("BUFF".PROCESS <= 15);
END_REGION

REGION Network 26
   RUNG wire#powerrail
      Contact( "AlwaysTRUE" )
      wire#w1
      I_Contact( "IO BITS"."JACKET SAFETY BIT" )
      S_Coil( "AUXILIARY"."PWD STEAM ON" )
   END_RUNG
   RUNG wire#w1
      Contact( "IO BITS"."JACKET SAFETY BIT" )
      R_Coil( "AUXILIARY"."PWD STEAM ON" )
   END_RUNG
   RUNG wire#w1
      Sub(in1 := "RETAIN"."SET PWD TEMP", in2 := "RETAIN"."SET CONTROL BAND", out => "PWD TEMP ON")
   END_RUNG
   // the same network as SCL:
   IF "AlwaysTRUE" AND NOT "IO BITS"."JACKET SAFETY BIT" THEN "AUXILIARY"."PWD STEAM ON" := TRUE; END_IF;
   IF "AlwaysTRUE" AND "IO BITS"."JACKET SAFETY BIT" THEN "AUXILIARY"."PWD STEAM ON" := FALSE; END_IF;
   IF "AlwaysTRUE" THEN "PWD TEMP ON" := "RETAIN"."SET PWD TEMP" - "RETAIN"."SET CONTROL BAND"; END_IF;
END_REGION

REGION Network 27
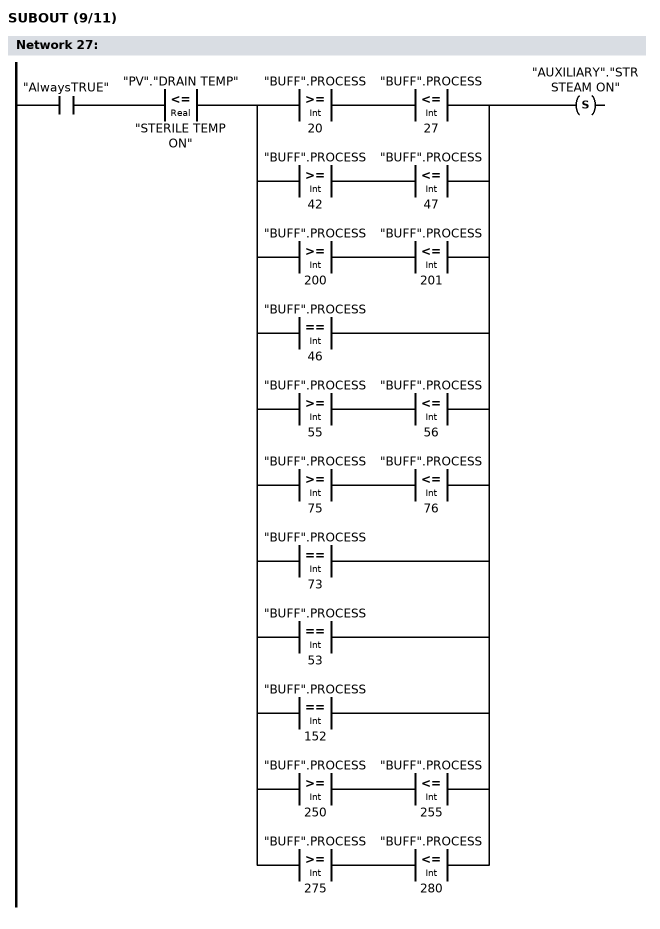
   RUNG wire#powerrail
      Contact( "AlwaysTRUE" )
      { S7_Templates := "SrcType := Real" } LE_Contact(in1 := "PV"."DRAIN TEMP", in2 := "STERILE TEMP ON")
      wire#w1
      { S7_Templates := "SrcType := Int" } GE_Contact(in1 := "BUFF".PROCESS, in2 := 20)
      { S7_Templates := "SrcType := Int" } LE_Contact(in1 := "BUFF".PROCESS, in2 := 27)
      wire#w2
      S_Coil( "AUXILIARY"."STR STEAM ON" )
   END_RUNG
   RUNG wire#w1
      { S7_Templates := "SrcType := Int" } GE_Contact(in1 := "BUFF".PROCESS, in2 := 42)
      { S7_Templates := "SrcType := Int" } LE_Contact(in1 := "BUFF".PROCESS, in2 := 47)
   END_RUNG wire#w2
   RUNG wire#w1
      { S7_Templates := "SrcType := Int" } GE_Contact(in1 := "BUFF".PROCESS, in2 := 200)
      { S7_Templates := "SrcType := Int" } LE_Contact(in1 := "BUFF".PROCESS, in2 := 201)
   END_RUNG wire#w2
   RUNG wire#w1
      { S7_Templates := "SrcType := Int" } EQ_Contact(in1 := "BUFF".PROCESS, in2 := 46)
   END_RUNG wire#w2
   RUNG wire#w1
      { S7_Templates := "SrcType := Int" } GE_Contact(in1 := "BUFF".PROCESS, in2 := 55)
      { S7_Templates := "SrcType := Int" } LE_Contact(in1 := "BUFF".PROCESS, in2 := 56)
   END_RUNG wire#w2
   RUNG wire#w1
      { S7_Templates := "SrcType := Int" } GE_Contact(in1 := "BUFF".PROCESS, in2 := 75)
      { S7_Templates := "SrcType := Int" } LE_Contact(in1 := "BUFF".PROCESS, in2 := 76)
   END_RUNG wire#w2
   RUNG wire#w1
      { S7_Templates := "SrcType := Int" } EQ_Contact(in1 := "BUFF".PROCESS, in2 := 73)
   END_RUNG wire#w2
   RUNG wire#w1
      { S7_Templates := "SrcType := Int" } EQ_Contact(in1 := "BUFF".PROCESS, in2 := 53)
   END_RUNG wire#w2
   RUNG wire#w1
      { S7_Templates := "SrcType := Int" } EQ_Contact(in1 := "BUFF".PROCESS, in2 := 152)
   END_RUNG wire#w2
   RUNG wire#w1
      { S7_Templates := "SrcType := Int" } GE_Contact(in1 := "BUFF".PROCESS, in2 := 250)
      { S7_Templates := "SrcType := Int" } LE_Contact(in1 := "BUFF".PROCESS, in2 := 255)
   END_RUNG wire#w2
   RUNG wire#w1
      { S7_Templates := "SrcType := Int" } GE_Contact(in1 := "BUFF".PROCESS, in2 := 275)
      { S7_Templates := "SrcType := Int" } LE_Contact(in1 := "BUFF".PROCESS, in2 := 280)
   END_RUNG wire#w2
   // the same network as SCL:
   IF "AlwaysTRUE" AND ("PV"."DRAIN TEMP" <= "STERILE TEMP ON") AND ((("BUFF".PROCESS >= 20) AND ("BUFF".PROCESS <= 27)) OR (("BUFF".PROCESS >= 42) AND ("BUFF".PROCESS <= 47)) OR (("BUFF".PROCESS >= 200) AND ("BUFF".PROCESS <= 201)) OR ("BUFF".PROCESS = 46) OR (("BUFF".PROCESS >= 55) AND ("BUFF".PROCESS <= 56)) OR (("BUFF".PROCESS >= 75) AND ("BUFF".PROCESS <= 76)) OR ("BUFF".PROCESS = 73) OR ("BUFF".PROCESS = 53) OR ("BUFF".PROCESS = 152) OR (("BUFF".PROCESS >= 250) AND ("BUFF".PROCESS <= 255)) OR (("BUFF".PROCESS >= 275) AND ("BUFF".PROCESS <= 280))) THEN
       "AUXILIARY"."STR STEAM ON" := TRUE;
   END_IF;
END_REGION

REGION Network 28
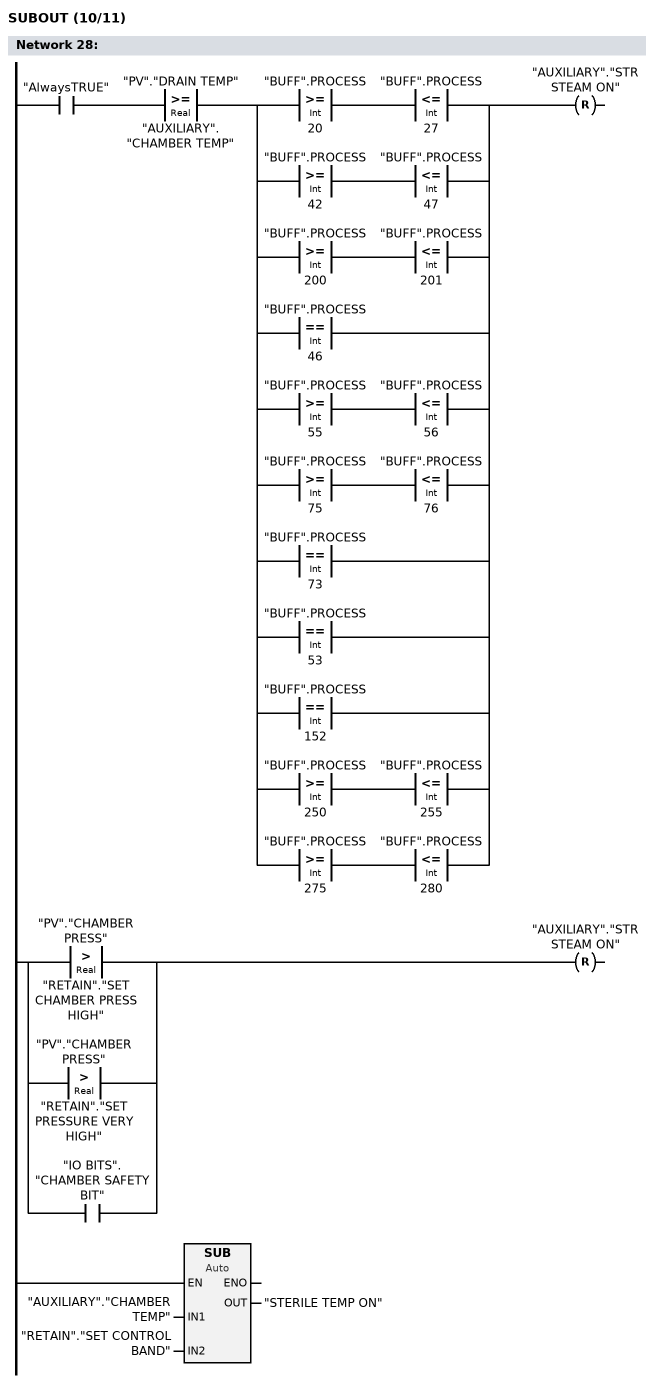
   RUNG wire#powerrail
      Contact( "AlwaysTRUE" )
      { S7_Templates := "SrcType := Real" } GE_Contact(in1 := "PV"."DRAIN TEMP", in2 := "AUXILIARY"."CHAMBER TEMP")
      wire#w1
      { S7_Templates := "SrcType := Int" } GE_Contact(in1 := "BUFF".PROCESS, in2 := 20)
      { S7_Templates := "SrcType := Int" } LE_Contact(in1 := "BUFF".PROCESS, in2 := 27)
      wire#w2
      R_Coil( "AUXILIARY"."STR STEAM ON" )
   END_RUNG
   RUNG wire#w1
      { S7_Templates := "SrcType := Int" } GE_Contact(in1 := "BUFF".PROCESS, in2 := 42)
      { S7_Templates := "SrcType := Int" } LE_Contact(in1 := "BUFF".PROCESS, in2 := 47)
   END_RUNG wire#w2
   RUNG wire#w1
      { S7_Templates := "SrcType := Int" } GE_Contact(in1 := "BUFF".PROCESS, in2 := 200)
      { S7_Templates := "SrcType := Int" } LE_Contact(in1 := "BUFF".PROCESS, in2 := 201)
   END_RUNG wire#w2
   RUNG wire#w1
      { S7_Templates := "SrcType := Int" } EQ_Contact(in1 := "BUFF".PROCESS, in2 := 46)
   END_RUNG wire#w2
   RUNG wire#w1
      { S7_Templates := "SrcType := Int" } GE_Contact(in1 := "BUFF".PROCESS, in2 := 55)
      { S7_Templates := "SrcType := Int" } LE_Contact(in1 := "BUFF".PROCESS, in2 := 56)
   END_RUNG wire#w2
   RUNG wire#w1
      { S7_Templates := "SrcType := Int" } GE_Contact(in1 := "BUFF".PROCESS, in2 := 75)
      { S7_Templates := "SrcType := Int" } LE_Contact(in1 := "BUFF".PROCESS, in2 := 76)
   END_RUNG wire#w2
   RUNG wire#w1
      { S7_Templates := "SrcType := Int" } EQ_Contact(in1 := "BUFF".PROCESS, in2 := 73)
   END_RUNG wire#w2
   RUNG wire#w1
      { S7_Templates := "SrcType := Int" } EQ_Contact(in1 := "BUFF".PROCESS, in2 := 53)
   END_RUNG wire#w2
   RUNG wire#w1
      { S7_Templates := "SrcType := Int" } EQ_Contact(in1 := "BUFF".PROCESS, in2 := 152)
   END_RUNG wire#w2
   RUNG wire#w1
      { S7_Templates := "SrcType := Int" } GE_Contact(in1 := "BUFF".PROCESS, in2 := 250)
      { S7_Templates := "SrcType := Int" } LE_Contact(in1 := "BUFF".PROCESS, in2 := 255)
   END_RUNG wire#w2
   RUNG wire#w1
      { S7_Templates := "SrcType := Int" } GE_Contact(in1 := "BUFF".PROCESS, in2 := 275)
      { S7_Templates := "SrcType := Int" } LE_Contact(in1 := "BUFF".PROCESS, in2 := 280)
   END_RUNG wire#w2
   RUNG wire#powerrail
      { S7_Templates := "SrcType := Real" } GT_Contact(in1 := "PV"."CHAMBER PRESS", in2 := "RETAIN"."SET CHAMBER PRESS HIGH")
      wire#w3
      R_Coil( "AUXILIARY"."STR STEAM ON" )
   END_RUNG
   RUNG wire#powerrail
      { S7_Templates := "SrcType := Real" } GT_Contact(in1 := "PV"."CHAMBER PRESS", in2 := "RETAIN"."SET PRESSURE VERY HIGH")
   END_RUNG wire#w3
   RUNG wire#powerrail
      Contact( "IO BITS"."CHAMBER SAFETY BIT" )
   END_RUNG wire#w3
   RUNG wire#powerrail
      Sub(in1 := "AUXILIARY"."CHAMBER TEMP", in2 := "RETAIN"."SET CONTROL BAND", out => "STERILE TEMP ON")
   END_RUNG
   // the same network as SCL:
   IF "AlwaysTRUE" AND ("PV"."DRAIN TEMP" >= "AUXILIARY"."CHAMBER TEMP") AND ((("BUFF".PROCESS >= 20) AND ("BUFF".PROCESS <= 27)) OR (("BUFF".PROCESS >= 42) AND ("BUFF".PROCESS <= 47)) OR (("BUFF".PROCESS >= 200) AND ("BUFF".PROCESS <= 201)) OR ("BUFF".PROCESS = 46) OR (("BUFF".PROCESS >= 55) AND ("BUFF".PROCESS <= 56)) OR (("BUFF".PROCESS >= 75) AND ("BUFF".PROCESS <= 76)) OR ("BUFF".PROCESS = 73) OR ("BUFF".PROCESS = 53) OR ("BUFF".PROCESS = 152) OR (("BUFF".PROCESS >= 250) AND ("BUFF".PROCESS <= 255)) OR (("BUFF".PROCESS >= 275) AND ("BUFF".PROCESS <= 280))) THEN
       "AUXILIARY"."STR STEAM ON" := FALSE;
   END_IF;
   IF ("PV"."CHAMBER PRESS" > "RETAIN"."SET CHAMBER PRESS HIGH") OR ("PV"."CHAMBER PRESS" > "RETAIN"."SET PRESSURE VERY HIGH") OR "IO BITS"."CHAMBER SAFETY BIT" THEN
       "AUXILIARY"."STR STEAM ON" := FALSE;
   END_IF;
   "STERILE TEMP ON" := "AUXILIARY"."CHAMBER TEMP" - "RETAIN"."SET CONTROL BAND";
END_REGION

REGION Network 29
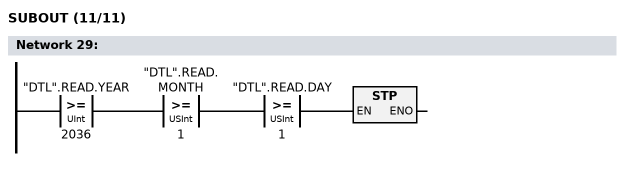
   RUNG wire#powerrail
      { S7_Templates := "SrcType := UInt" } GE_Contact(in1 := "DTL".READ.YEAR, in2 := 2036)
      { S7_Templates := "SrcType := USInt" } GE_Contact(in1 := "DTL".READ.MONTH, in2 := 1)
      { S7_Templates := "SrcType := USInt" } GE_Contact(in1 := "DTL".READ.DAY, in2 := 1)
      STP()
   END_RUNG
   // the same network as SCL:
   IF ("DTL".READ.YEAR >= 2036) AND ("DTL".READ.MONTH >= 1) AND ("DTL".READ.DAY >= 1) THEN STP(); END_IF;
END_REGION
END_FUNCTION
